FUNCTION_BLOCK FB_EventMessage 
VAR_INPUT 
	bEvent			: BOOL; 
	nEventID		: UDINT; 
	sSource			: STRING; 
END_VAR 
VAR_OUTPUT 
END_VAR 
VAR
	bIsInitalized : BOOL;
	
	fbSourceInfo 	: FB_TcSourceInfo;
	fbMessage 		: FB_TcMessage;
	eventEntry 		: TcEventEntry;
	fbRtEvent		: R_TRIG;
	hr 				: HRESULT;
	hrLastError		: HRESULT;
	
END_VAR

// initialization 
	IF NOT bIsInitalized THEN
		bIsInitalized:= TRUE;
		
		IF nEventID> 16#04FF THEN
			eventEntry:= Tc_Events.myWarningEventClass.x0500; 
		ELSE
			eventEntry:= TC_Events.myInfoEventClass.x0000; 
		END_IF
		
		eventEntry.nEventId:= nEventID;
		fbSourceInfo.Clear(); 
		fbSourceInfo.sName := sSource;
		
		hr:= fbMessage.CreateEx(eventEntry, ipSourceInfo:= fbSourceInfo); 
		IF FAILED (hr) THEN
			hrLastError:= hr; 
		END_IF 
	END_IF
	
// event trigger 
	fbRtEvent (CLK:= bEvent);

// message sent
	IF fbRtEvent.Q THEN
		hr:= fbMessage. Send(0); 
		IF FAILED (hr) THEN
			hrLastError:= hr;
		END_IF 
	END_IF

END_FUNCTION_BLOCK

(* stored: Version 1.1.0.1, ProductVersion 3.1.4024.11
   POU FB_EventMessage: Id {5fc64599-ad83-4f07-975f-6d21140eb252}, SpecialFunc None *)
